# EPICS autosave request: iocBoot/obsolete/ioc13ida_E_Mono_PMAC/auto_positions.req
file "CARS_motor_positions.req",         P=$(P), M=m73
file "CARS_motor_positions.req",         P=$(P), M=m74
file "CARS_motor_positions.req",         P=$(P), M=m75
file "CARS_motor_positions.req",         P=$(P), M=m76
file "CARS_motor_positions.req",         P=$(P), M=m77
file "CARS_motor_positions.req",         P=$(P), M=m78
file "CARS_motor_positions.req",         P=$(P), M=m79
file "CARS_motor_positions.req",         P=$(P), M=m80
file "CARS_motor_positions.req",         P=$(P), M=m81
